// TIA Portal V18 export
FUNCTION "AHURoomSPTarget" : Void   // FC60006, LAD
{ S7_Optimized_Access := 'TRUE' }
VERSION : 0.1
// stored: AutoNumber false, IsIECCheckEnabled false, SetENOAutomatically false, UDAEnableTagReadback false
   VAR_INPUT
      iUnitID : Int;
      rActualStoreSPTempHeating : Real;
      rActualStoreSPTempCooling : Real;
      rActualStoreSPIAQ : Real;
      rActualStoreSPdP : Real;
      rAHUShiftTempHeatingSP : Real;
      rAHUShiftTempCoolingSP : Real;
      rAHUShiftIAQSP : Real;
      rAHUShiftdPSP : Real;
   END_VAR
   VAR_OUTPUT
      rTargetAHUTempHeatingSP : Real;
      rTargetAHUTempCoolingSP : Real;
      rTargetAHUIAQSP : Real;
      rTargetAHUdPSP : Real;
   END_VAR
   VAR_TEMP
      iTargetUnitMode_old : Int;
      xResetActualOperationMode : Bool;
      iActualUnitMode_old : Int;
      xResetTargetSetpoints : Bool;
   END_VAR
BEGIN

REGION Network 1 (SCL)
   #rTargetAHUTempHeatingSP := #rActualStoreSPTempHeating + #rAHUShiftTempHeatingSP;
   #rTargetAHUTempCoolingSP := #rActualStoreSPTempCooling + #rAHUShiftTempCoolingSP;
   #rTargetAHUIAQSP := #rActualStoreSPIAQ + #rAHUShiftIAQSP;
   #rTargetAHUdPSP := #rActualStoreSPdP + #rAHUShiftdPSP;
END_REGION
END_FUNCTION
